// TIA Portal V21 export
DATA_BLOCK "Tema"   // DB34
{ S7_Optimized_Access := 'TRUE' }
// stored: MemoryReserve 100
   VAR
      TemaAttuale : Int := 0;
   END_VAR
BEGIN
END_DATA_BLOCK
